LIN {X 0,Y 36.224,Z 815.915,A -85,B 0,C 180,E1 -30099.101,E2 -30099.101} C_VEL
LIN {X 0,Y 29.533,Z 814.07,A -85,B 0,C 180,E1 -30121.58,E2 -30121.58} C_VEL
LIN {X 0,Y 28.318,Z 811.531,A -85,B 0,C 180,E1 -30143.088,E2 -30143.088} C_VEL
LIN {X 0,Y 30.715,Z 808.057,A -85,B 0,C 180,E1 -30163.227,E2 -30163.227} C_VEL
LIN {X 0,Y 32.06,Z 806.772,A -85,B 0,C 180,E1 -30168.532,E2 -30168.532} C_VEL
LIN {X 0,Y 31.122,Z 805.787,A -85,B 0,C 180,E1 -30175.405,E2 -30175.405} C_VEL
LIN {X 0,Y 28.185,Z 803.303,A -85,B 0,C 180,E1 -30201.923,E2 -30201.923} C_VEL
LIN {X 0,Y 31.507,Z 808.669,A -85,B 0,C 180,E1 -30223.118,E2 -30223.118} C_VEL
LIN {X 0,Y 38.845,Z 813.205,A -85,B 0,C 180,E1 -30240,E2 -30240} C_VEL
LIN {X 0,Y 50.41,Z 816.923,A -85,B 0,C 180,E1 -30252.605,E2 -30252.605} C_VEL
LIN {X 0,Y 59.179,Z 818.511,A -85,B 0,C 180,E1 -30258.187,E2 -30258.187} C_VEL
LIN {X 0,Y 60.011,Z 818.796,A -85,B 0,C 180,E1 -30260.468,E2 -30260.468} C_VEL
LIN {X 0,Y 47.956,Z 817.889,A -85,B 0,C 180,E1 -30268.444,E2 -30268.444} C_VEL
LIN {X 0,Y 37.652,Z 815.699,A -85,B 0,C 180,E1 -30281.703,E2 -30281.703} C_VEL
LIN {X 0,Y 31.161,Z 812.419,A -85,B 0,C 180,E1 -30302.279,E2 -30302.279} C_VEL
LIN {X 0,Y 29.102,Z 815.053,A -85,B 0,C 180,E1 -30316.026,E2 -30316.026} C_VEL
LIN {X 0,Y 28.638,Z 817.011,A -85,B 0,C 180,E1 -30330,E2 -30330} C_VEL
LIN {X 0,Y 28.501,Z 818.405,A -85,B 0,C 180,E1 -30344.276,E2 -30344.276} C_VEL
LIN {X 0,Y 29.997,Z 819.387,A -85,B 0,C 180,E1 -30357.942,E2 -30357.942} C_VEL
LIN {X 0,Y 37.183,Z 820.133,A -85,B 0,C 180,E1 -30379.116,E2 -30379.116} C_VEL
LIN {X 0,Y 47.741,Z 819.394,A -85,B 0,C 180,E1 -30392.035,E2 -30392.035} C_VEL
LIN {X 0,Y 59.859,Z 817.048,A -85,B 0,C 180,E1 -30399.925,E2 -30399.925} C_VEL
LIN {X 0,Y 69.51,Z 814.247,A -85,B 0,C 180,E1 -30403.843,E2 -30403.843} C_VEL
LIN {X 0,Y 79.441,Z 810.463,A -85,B 0,C 180,E1 -30406.685,E2 -30406.685} C_VEL
LIN {X 0,Y 89.543,Z 805.585,A -85,B 0,C 180,E1 -30408.833,E2 -30408.833} C_VEL
LIN {X 0,Y 99.775,Z 799.472,A -85,B 0,C 180,E1 -30410.442,E2 -30410.442} C_VEL
LIN {X 0,Y 110.091,Z 791.92,A -85,B 0,C 180,E1 -30411.674,E2 -30411.674} C_VEL
LIN {X 0,Y 120.445,Z 782.472,A -85,B 0,C 180,E1 -30412.716,E2 -30412.716} C_VEL
LIN {X 0,Y 129.144,Z 772.744,A -85,B 0,C 180,E1 -30413.284,E2 -30413.284} C_VEL
LIN {X 0,Y 136.977,Z 761.885,A -85,B 0,C 180,E1 -30413.756,E2 -30413.756} C_VEL
LIN {X 0,Y 143.643,Z 750.191,A -85,B 0,C 180,E1 -30414.119,E2 -30414.119} C_VEL
LIN {X 0,Y 144.17,Z 749.151,A -85,B 0,C 180,E1 -30414.145,E2 -30414.145} C_VEL
LIN {X 0,Y 145.036,Z 747.315,A -85,B 0,C 180,E1 -30414.438,E2 -30414.438} C_VEL
LIN {X 0,Y 145.002,Z 747.267,A -85,B 0,C 180,E1 -30415.363,E2 -30415.363} C_VEL
LIN {X 0,Y 144.395,Z 748.488,A -85,B 0,C 180,E1 -30415.779,E2 -30415.779} C_VEL
LIN {X 0,Y 138.174,Z 759.621,A -85,B 0,C 180,E1 -30416.514,E2 -30416.514} C_VEL
LIN {X 0,Y 130.915,Z 769.994,A -85,B 0,C 180,E1 -30417.387,E2 -30417.387} C_VEL
LIN {X 0,Y 123.038,Z 779.157,A -85,B 0,C 180,E1 -30418.342,E2 -30418.342} C_VEL
LIN {X 0,Y 114.205,Z 787.545,A -85,B 0,C 180,E1 -30419.567,E2 -30419.567} C_VEL
LIN {X 0,Y 111.959,Z 789.431,A -85,B 0,C 180,E1 -30419.917,E2 -30419.917} C_VEL
LIN {X 0,Y 107.358,Z 793.085,A -85,B 0,C 180,E1 -30420.284,E2 -30420.284} C_VEL
LIN {X 0,Y 99.192,Z 798.709,A -85,B 0,C 180,E1 -30420.006,E2 -30420.006} C_VEL
LIN {X 0,Y 90.611,Z 803.633,A -85,B 0,C 180,E1 -30419.734,E2 -30419.734} C_VEL
LIN {X 0,Y 85.359,Z 806.186,A -85,B 0,C 180,E1 -30420.277,E2 -30420.277} C_VEL
LIN {X 0,Y 73.882,Z 810.755,A -85,B 0,C 180,E1 -30422.822,E2 -30422.822} C_VEL
LIN {X 0,Y 61.782,Z 814.182,A -85,B 0,C 180,E1 -30426.532,E2 -30426.532} C_VEL
LIN {X 0,Y 50.248,Z 816.149,A -85,B 0,C 180,E1 -30431.75,E2 -30431.75} C_VEL
LIN {X 0,Y 37.766,Z 816.873,A -85,B 0,C 180,E1 -30441.498,E2 -30441.498} C_VEL
LIN {X 0,Y 32.136,Z 816.586,A -85,B 0,C 180,E1 -30448.984,E2 -30448.984} C_VEL
LIN {X 0,Y 23.412,Z 814.812,A -85,B 0,C 180,E1 -30473.104,E2 -30473.104} C_VEL
LIN {X 0,Y 21.226,Z 812.082,A -85,B 0,C 180,E1 -30503.363,E2 -30503.363} C_VEL
LIN {X 0,Y 23.776,Z 808.937,A -85,B 0,C 180,E1 -30527.193,E2 -30527.193} C_VEL
LIN {X 0,Y 24.243,Z 808.028,A -85,B 0,C 180,E1 -30533.415,E2 -30533.415} C_VEL
LIN {X 0,Y 22.358,Z 805.138,A -85,B 0,C 180,E1 -30576.12,E2 -30576.12} C_VEL
LIN {X 0,Y 29.138,Z 810.579,A -85,B 0,C 180,E1 -30600,E2 -30600} C_VEL
LIN {X 0,Y 40.432,Z 815.29,A -85,B 0,C 180,E1 -30615.119,E2 -30615.119} C_VEL
LIN {X 0,Y 44.616,Z 816.481,A -85,B 0,C 180,E1 -30618.363,E2 -30618.363} C_VEL
LIN {X 0,Y 45.022,Z 816.74,A -85,B 0,C 180,E1 -30620.513,E2 -30620.513} C_VEL
LIN {X 0,Y 33.414,Z 814.271,A -85,B 0,C 180,E1 -30632.721,E2 -30632.721} C_VEL
LIN {X 0,Y 25.677,Z 811.086,A -85,B 0,C 180,E1 -30652.607,E2 -30652.607} C_VEL
LIN {X 0,Y 22.29,Z 814.233,A -85,B 0,C 180,E1 -30671.621,E2 -30671.621} C_VEL
LIN {X 0,Y 21.546,Z 816.227,A -85,B 0,C 180,E1 -30690,E2 -30690} C_VEL
LIN {X 0,Y 21.679,Z 817.652,A -85,B 0,C 180,E1 -30708.916,E2 -30708.916} C_VEL
LIN {X 0,Y 23.927,Z 818.676,A -85,B 0,C 180,E1 -30725.975,E2 -30725.975} C_VEL
LIN {X 0,Y 32.954,Z 819.508,A -85,B 0,C 180,E1 -30748.544,E2 -30748.544} C_VEL
LIN {X 0,Y 44.838,Z 818.842,A -85,B 0,C 180,E1 -30760.124,E2 -30760.124} C_VEL
LIN {X 0,Y 52.684,Z 817.64,A -85,B 0,C 180,E1 -30764.526,E2 -30764.526} C_VEL
LIN {X 0,Y 64.49,Z 814.872,A -85,B 0,C 180,E1 -30768.746,E2 -30768.746} C_VEL
LIN {X 0,Y 74.685,Z 811.495,A -85,B 0,C 180,E1 -30771.13,E2 -30771.13} C_VEL
LIN {X 0,Y 84.983,Z 807.073,A -85,B 0,C 180,E1 -30772.911,E2 -30772.911} C_VEL
LIN {X 0,Y 95.372,Z 801.488,A -85,B 0,C 180,E1 -30774.15,E2 -30774.15} C_VEL
LIN {X 0,Y 105.803,Z 794.556,A -85,B 0,C 180,E1 -30775.107,E2 -30775.107} C_VEL
LIN {X 0,Y 112.773,Z 788.993,A -85,B 0,C 180,E1 -30775.633,E2 -30775.633} C_VEL
LIN {X 0,Y 112.702,Z 788.993,A -85,B 0,C 180,E1 -30776.134,E2 -30776.134} C_VEL
LIN {X 0,Y 102,Z 796.957,A -85,B 0,C 180,E1 -30777.511,E2 -30777.511} C_VEL
LIN {X 0,Y 91.371,Z 803.245,A -85,B 0,C 180,E1 -30779.168,E2 -30779.168} C_VEL
LIN {X 0,Y 85.359,Z 806.186,A -85,B 0,C 180,E1 -30780.277,E2 -30780.277} C_VEL
LIN {X 0,Y 79.994,Z 808.527,A -85,B 0,C 180,E1 -30780.903,E2 -30780.903} C_VEL
LIN {X 0,Y 70.699,Z 811.994,A -85,B 0,C 180,E1 -30780.731,E2 -30780.731} C_VEL
LIN {X 0,Y 61.167,Z 814.688,A -85,B 0,C 180,E1 -30780.492,E2 -30780.492} C_VEL
LIN {X 0,Y 55.438,Z 815.772,A -85,B 0,C 180,E1 -30781.387,E2 -30781.387} C_VEL
LIN {X 0,Y 49.283,Z 816.682,A -85,B 0,C 180,E1 -30783.423,E2 -30783.423} C_VEL
LIN {X 0,Y 35.747,Z 817.475,A -85,B 0,C 180,E1 -30790.578,E2 -30790.578} C_VEL
LIN {X 0,Y 29.307,Z 817.258,A -85,B 0,C 180,E1 -30796.422,E2 -30796.422} C_VEL
LIN {X 0,Y 18.156,Z 815.548,A -85,B 0,C 180,E1 -30819.273,E2 -30819.273} C_VEL
LIN {X 0,Y 14.14,Z 812.641,A -85,B 0,C 180,E1 -30863.755,E2 -30863.755} C_VEL
LIN {X 0,Y 15.376,Z 811.067,A -85,B 0,C 180,E1 -30883.211,E2 -30883.211} C_VEL
LIN {X 0,Y 16.533,Z 809.883,A -85,B 0,C 180,E1 -30895.155,E2 -30895.155} C_VEL
LIN {X 0,Y 19.131,Z 806.98,A -85,B 0,C 180,E1 -30959.411,E2 -30959.411} C_VEL
LIN {X 0,Y 29.6,Z 812.404,A -85,B 0,C 180,E1 -30978.248,E2 -30978.248} C_VEL
LIN {X 0,Y 30.21,Z 812.808,A -85,B 0,C 180,E1 -30981.481,E2 -30981.481} C_VEL
LIN {X 0,Y 21.301,Z 809.753,A -85,B 0,C 180,E1 -30998.411,E2 -30998.411} C_VEL
LIN {X 0,Y 15.715,Z 813.393,A -85,B 0,C 180,E1 -31023.436,E2 -31023.436} C_VEL
LIN {X 0,Y 14.453,Z 815.442,A -85,B 0,C 180,E1 -31050,E2 -31050} C_VEL
LIN {X 0,Y 18.64,Z 817.956,A -85,B 0,C 180,E1 -31098.943,E2 -31098.943} C_VEL
LIN {X 0,Y 23.846,Z 818.63,A -85,B 0,C 180,E1 -31112.148,E2 -31112.148} C_VEL
LIN {X 0,Y 36.296,Z 818.771,A -85,B 0,C 180,E1 -31125.495,E2 -31125.495} C_VEL
LIN {X 0,Y 49.71,Z 817.418,A -85,B 0,C 180,E1 -31131.746,E2 -31131.746} C_VEL
LIN {X 0,Y 63.486,Z 814.448,A -85,B 0,C 180,E1 -31135.06,E2 -31135.06} C_VEL
LIN {X 0,Y 70.437,Z 812.367,A -85,B 0,C 180,E1 -31136.152,E2 -31136.152} C_VEL
LIN {X 0,Y 74.081,Z 811.039,A -85,B 0,C 180,E1 -31137.13,E2 -31137.13} C_VEL
LIN {X 0,Y 63.255,Z 814.169,A -85,B 0,C 180,E1 -31139.3,E2 -31139.3} C_VEL
LIN {X 0,Y 55.438,Z 815.772,A -85,B 0,C 180,E1 -31141.387,E2 -31141.387} C_VEL
LIN {X 0,Y 49.664,Z 816.688,A -85,B 0,C 180,E1 -31142.487,E2 -31142.487} C_VEL
LIN {X 0,Y 39.79,Z 817.699,A -85,B 0,C 180,E1 -31142.493,E2 -31142.493} C_VEL
LIN {X 0,Y 31.851,Z 817.948,A -85,B 0,C 180,E1 -31142.214,E2 -31142.214} C_VEL
LIN {X 0,Y 25.976,Z 817.747,A -85,B 0,C 180,E1 -31143.521,E2 -31143.521} C_VEL
LIN {X 0,Y 24.076,Z 817.559,A -85,B 0,C 180,E1 -31144.686,E2 -31144.686} C_VEL
LIN {X 0,Y 14.679,Z 816.288,A -85,B 0,C 180,E1 -31156.762,E2 -31156.762} C_VEL
LIN {X 0,Y 9.067,Z 814.873,A -85,B 0,C 180,E1 -31179.185,E2 -31179.185} C_VEL
LIN {X 0,Y 7.157,Z 813.004,A -85,B 0,C 180,E1 -31230,E2 -31230} C_VEL
LIN {X 0,Y 8.561,Z 811.577,A -85,B 0,C 180,E1 -31264.826,E2 -31264.826} C_VEL
LIN {X 0,Y 14.637,Z 809.637,A -85,B 0,C 180,E1 -31336.204,E2 -31336.204} C_VEL
LIN {X 0,Y 15.422,Z 809.921,A -85,B 0,C 180,E1 -31344.299,E2 -31344.299} C_VEL
LIN {X 0,Y 9.498,Z 812.763,A -85,B 0,C 180,E1 -31367.724,E2 -31367.724} C_VEL
LIN {X 0,Y 7.361,Z 814.658,A -85,B 0,C 180,E1 -31410,E2 -31410} C_VEL
LIN {X 0,Y 14.963,Z 817.236,A -85,B 0,C 180,E1 -31479.947,E2 -31479.947} C_VEL
LIN {X 0,Y 21.459,Z 817.948,A -85,B 0,C 180,E1 -31489.266,E2 -31489.266} C_VEL
LIN {X 0,Y 28.262,Z 818.26,A -85,B 0,C 180,E1 -31494.076,E2 -31494.076} C_VEL
LIN {X 0,Y 35.194,Z 818.18,A -85,B 0,C 180,E1 -31496.809,E2 -31496.809} C_VEL
LIN {X 0,Y 35.146,Z 818.078,A -85,B 0,C 180,E1 -31498.825,E2 -31498.825} C_VEL
LIN {X 0,Y 24.076,Z 817.559,A -85,B 0,C 180,E1 -31504.686,E2 -31504.686} C_VEL
LIN {X 0,Y 19.375,Z 817.138,A -85,B 0,C 180,E1 -31507.432,E2 -31507.432} C_VEL
LIN {X 0,Y 11.333,Z 816.108,A -85,B 0,C 180,E1 -31508.729,E2 -31508.729} C_VEL
LIN {X 0,Y 1.646,Z 814.239,A -85,B 0,C 180,E1 -31505.798,E2 -31505.798} C_VEL
LIN {X 0,Y 1.528,Z 813.39,A -85,B 0,C 180,E1 -31680.001,E2 -31680.001} C_VEL
LIN {X 0,Y 1.852,Z 813.296,A -85,B 0,C 180,E1 -31680.001,E2 -31680.001} C_VEL
LIN {X 0,Y 0.079,Z 813.84,A -85,B 0,C 180,E1 -31770,E2 -31770} C_VEL
LIN {X 0,Y 1.528,Z 813.39,A -85,B 0,C 180,E1 -31680.001,E2 -31680.001} C_VEL
LIN {X 0,Y 1.528,Z 813.39,A -85,B 0,C 180,E1 -31680.001,E2 -31680.001}

QRS_NEXT_CUT()

QRS_NEXT()
QRS_HOME()

END
